{attribute 'GeneratedUsingTerminal: EL3773-0000-0016'}
{attribute addProperty BoxType "EL3773-0000-0016"}
{attribute addProperty Id "U1_STATUSAT %I*U1_STATUS_B07533568"}
{attribute addProperty CRC "2018444205"}
{attribute addProperty Size "8"}
TYPE L1_Voltage_Status_784F03AD :
STRUCT
	{attribute addProperty Name "U1_STATUS"}
	U1_STATUS AT %I* : U1_STATUS_B0753356;
END_STRUCT
END_TYPE

(* stored: Version 1.2.0.0, ProductVersion 3.1.4024.9
   DUT L1_Voltage_Status_784F03AD: Id {42dd7a68-5c56-4e67-af90-7d94a2933487} *)
